FUNCTION_BLOCK CheckStatusVanHetSysteem
VAR
	//Defenieren van de Xas en functies om deze te manipuleren
	XasDrive: AXIS_REF;
	XasDrivePower: MC_Power;
	DePositieVanDeXas AT %I* : LREAL;
	StopDeBoot : MC_Stop;
	VeranderDriveOperationMode : MC_WriteDriveOperationMode;
	OutDeurslot   AT %Q* : BOOL;
	
	//Inputs Vanuit HMI en Variabele voor checken van drive status
	StatusVanDePower : (Uit, Actief, Error );
	KnopDriveAan2 AT %I* : BOOL;
	KnopDriveUit  AT %I* : BOOL;
	IndicatieDriveIsActief   AT %Q* : BOOL;
	KnopStopKnop AT %I* : BOOL;	
	KnopDoorgaan AT %I* : BOOL;	
	
	//Variabele voor het bepalen van de state van het systeem
	StatusVanDeStateVanHetSysteem : (Uit, Joggen, Locatie, Torque);
	KnopJoggModus AT %I* : BOOL;
	KnopLocatieModus  AT %I* : BOOL;
	KnopTorqueControl AT %I* : BOOL;
	IndicatieStatusIsUit   AT %Q* : BOOL;
	IndicatieStatusIsJoggen   AT %Q* : BOOL;
	IndicatieStatusIsLocatie   AT %Q* : BOOL;
	IndicatieStatusIsTorque   AT %Q* : BOOL;
	
	// variabele voor Jogg state
	XasJoggModusFB : MC_MoveVelocity;
	HetTypeJog : (LinksTraag, LinksSnel, RechtsSnel, RechtsTraag, StilStaan);
	KnopJoggModusLinksTraag AT %I* : BOOL;
	KnopJoggModusLinksSnel AT %I* : BOOL;
	KnopJoggModusRechtsTraag AT %I* : BOOL;
	KnopJoggModusRechtsSnel AT %I* : BOOL;
	
	// Variabele voor Locatie state
	XasLocatieModeFB : MC_MoveAbsolute;
	StatusLocatieStatemachine : (WachtenOpNieuweLocatie, Uitvoeren, Bezig, Klaar,Pauzen);
 	DeIngevoerdeTargetPositie AT %I* : LREAL;
	NogAfTeLeggenAfstand AT %Q* : LREAL;
	KnopLocatieUitvoeren AT %I* : BOOL;
	KlaarMetBewegen : BOOL :=FALSE ;
	
	//Variabele voor Torque control
	StatusTorqueStatemachine : (WachtenOpNieuwDoel, Bezig2, Stop);
	DOTorqueDing : MC_TorqueControl;
	DeIngevoerdeTorqueDoel AT %I* : LREAL;
	KnopHervatTorquecontrol AT %I* : BOOL;	
	
	// hoopelijk gelinkde I/O
	InputSensor1 AT %I* : BOOL;
	OutputSysteemIsActiefDeurslot AT %Q* : BOOL;
	SlotDicht: BOOL :=FALSE ;
	SlotOpen: BOOL :=TRUE ;
END_VAR

CheckDrivePower();
CheckStateVanHetSysteem();
	CASE StatusVanDeStateVanHetSysteem OF
		Uit:
			IndicatieStatusIsUit:=TRUE;
			IndicatieStatusIsJoggen:=FALSE;
			IndicatieStatusIsLocatie:=FALSE;
			IndicatieStatusIsTorque:=FALSE;
			OutputSysteemIsActiefDeurslot:=SlotDicht;
		Joggen:
			IndicatieStatusIsUit:=FALSE;
			IndicatieStatusIsJoggen:=TRUE;
			IndicatieStatusIsLocatie:=FALSE;
			IndicatieStatusIsTorque:=FALSE;
			DoJogStatemachine();
			OutputSysteemIsActiefDeurslot:=SlotOpen;
		Locatie:
			NogAfTeLeggenAfstand:= DeIngevoerdeTargetPositie - DePositieVanDeXas;
			IndicatieStatusIsUit:=FALSE;
			IndicatieStatusIsJoggen:=FALSE;
			IndicatieStatusIsLocatie:=TRUE;
			IndicatieStatusIsTorque:=FALSE;
			DoLocatieStatemachine();
			OutputSysteemIsActiefDeurslot:=SlotDicht;		
		Torque:
			NogAfTeLeggenAfstand:= DeIngevoerdeTargetPositie - DePositieVanDeXas;
			IndicatieStatusIsUit:=FALSE;
			IndicatieStatusIsJoggen:=FALSE;
			IndicatieStatusIsLocatie:=FALSE;
			IndicatieStatusIsTorque:=TRUE;
			DoTorqueStatemachine();
			OutputSysteemIsActiefDeurslot:=SlotDicht;
	END_CASE

ACTION CheckDrivePower:
	XasDrivePower
	(
    Axis:= XasDrive,
    Enable:= FALSE,
    Enable_Positive:= TRUE,
    Enable_Negative:= TRUE,
    Override:= 100,
    BufferMode:= ,
    Options:= ,
    Status=> ,
    Busy=> ,
    Active=> ,
    Error=> ,
    ErrorID=> 
	);
//Power Inputs
IF KnopDriveAan2 THEN
	StatusVanDePower:= Actief;
	IndicatieDriveIsActief:=TRUE;
	SetPowerHighElkeKant();
	OutDeurslot:= TRUE;//Deur open
	
END_IF
IF NOT IndicatieDriveIsActief THEN
	StatusVanDePower:=Uit;
	SetPowerLow();
	OutDeurslot:= FALSE;// Deur gesloten
END_IF

//evtueel error checken
END_ACTION

ACTION CheckStateVanHetSysteem:

	VeranderDriveOperationMode
(	Execute:=FALSE,
	DriveOperationMode:=DriveOperationMode_Torque,
	Options:=,
	Axis:=XasDrive,
	Done=>,
	Busy=>,
	Error=>,
	ErrorID=>,);


IF KnopJoggModus AND NOT KnopLocatieModus AND IndicatieDriveIsActief AND NOT KnopTorqueControl THEN
	StatusVanDeStateVanHetSysteem:=Joggen;
	VeranderDriveOperationMode
(	Execute:=TRUE,
	DriveOperationMode:=DriveOperationMode_Default,
	Options:=,
	Axis:=XasDrive,
	Done=>,
	Busy=>,
	Error=>,
	ErrorID=>,);
END_IF

IF NOT KnopJoggModus AND NOT KnopLocatieModus AND IndicatieDriveIsActief AND KnopTorqueControl THEN
	StatusVanDeStateVanHetSysteem:=Torque;
	VeranderDriveOperationMode
(	Execute:=TRUE,
	DriveOperationMode:=DriveOperationMode_Torque,
	Options:=,
	Axis:=XasDrive,
	Done=>,
	Busy=>,
	Error=>,
	ErrorID=>,);

END_IF

IF NOT KnopJoggModus AND  KnopLocatieModus AND IndicatieDriveIsActief AND NOT KnopTorqueControl THEN
	StatusVanDeStateVanHetSysteem:=Locatie;
		
	VeranderDriveOperationMode
(	Execute:=TRUE,
	DriveOperationMode:=DriveOperationMode_Default,
	Options:=,
	Axis:=XasDrive,
	Done=>,
	Busy=>,
	Error=>,
	ErrorID=>,);
END_IF
IF NOT IndicatieDriveIsActief OR  NOT KnopJoggModus AND NOT KnopLocatieModus AND NOT KnopTorqueControl THEN
	StatusVanDeStateVanHetSysteem:=Uit;
	
	VeranderDriveOperationMode
(	Execute:=TRUE,
	DriveOperationMode:=DriveOperationMode_Default,
	Options:=,
	Axis:=XasDrive,
	Done=>,
	Busy=>,
	Error=>,
	ErrorID=>,);
END_IF
END_ACTION

ACTION DoJogStatemachine:
XasJoggModusFB
	(
    Axis:= XasDrive,
	Direction:= 1,
	Velocity :=0 ,
	Execute:=FALSE,
	Deceleration:=0,
	Acceleration :=0,
	Jerk:= ,
	BufferMode:= ,
	Options := ,
	InVelocity => ,
	Active => ,
	Busy => ,
	CommandAborted => ,
	Error => ,
	ErrorID => ,
	);
	
	IF KnopJoggModusLinksTraag THEN
		HetTypeJog:=LinksTraag;
	END_IF
	IF KnopJoggModusLinksSnel THEN
		HetTypeJog:=LinksSnel;
	END_IF
	IF KnopJoggModusRechtsTraag THEN
		HetTypeJog:=RechtsTraag;
	END_IF
	IF KnopJoggModusRechtsSnel THEN
		HetTypeJog:=RechtsSnel;
	END_IF
	IF NOT KnopJoggModusLinksTraag AND NOT KnopJoggModusLinksSnel AND NOT KnopJoggModusRechtsTraag AND NOT KnopJoggModusRechtsSnel THEN
		HetTypeJog:=StilStaan;
	END_IF
	
CASE HetTypeJog OF
	StilStaan:
XasJoggModusFB
(
	Axis:= XasDrive,
	Direction:= 1,
	Velocity :=0 ,
	Execute:=TRUE,
	Deceleration:=0,
	Acceleration :=0,
	Jerk:= ,
	BufferMode:= ,
	Options := ,
	InVelocity => ,
	Active => ,
	Busy => ,
	CommandAborted => ,
	Error => ,
	ErrorID => ,
	);
		LinksTraag:
XasJoggModusFB
(
    Axis:= XasDrive,
	Direction:= MC_Positive_Direction ,
	Velocity :=250 ,
	Execute:=TRUE,
	Deceleration:=0,
	Acceleration :=0,
	Jerk:= ,
	BufferMode:= ,
	Options := ,
	InVelocity => ,
	Active => ,
	Busy => ,
	CommandAborted => ,
	Error => ,
	ErrorID => ,
	);
		LinksSnel:
XasJoggModusFB
(
    Axis:= XasDrive,
	Direction:= MC_Positive_Direction ,
	Velocity :=500 ,
	Execute:=TRUE,
	Deceleration:=0,
	Acceleration :=0,
	Jerk:= ,
	BufferMode:= ,
	Options := ,
	InVelocity => ,
	Active => ,
	Busy => ,
	CommandAborted => ,
	Error => ,
	ErrorID => ,
	);
		RechtsSnel:
XasJoggModusFB
(
    Axis:= XasDrive,
	Direction:= MC_Negative_Direction,
	Velocity :=500 ,
	Execute:=TRUE,
	Deceleration:=0,
	Acceleration :=0,
	Jerk:= ,
	BufferMode:= ,
	Options := ,
	InVelocity => ,
	Active => ,
	Busy => ,
	CommandAborted => ,
	Error => ,
	ErrorID => ,
	);
	
	
	RechtsTraag:
XasJoggModusFB
(
    Axis:= XasDrive,
	Direction:= MC_Negative_Direction,
	Velocity :=250,
	Execute:=TRUE,
	Deceleration:=0,
	Acceleration :=0,
	Jerk:= ,
	BufferMode:= ,
	Options := ,
	InVelocity => ,
	Active => ,
	Busy => ,
	CommandAborted => ,
	Error => ,
	ErrorID => ,
	);

END_CASE
END_ACTION

ACTION DoLocatieStatemachine:

		XasLocatieModeFB
(   Axis:= XasDrive,
	Execute:=FALSE,
	Position := 0,
	Velocity :=0 ,
	Deceleration:=0,
	Acceleration :=0,
	Jerk:= ,
	BufferMode:= ,
	Options := ,
	Done => KlaarMetBewegen,
	Active => ,
	Busy => ,
	CommandAborted => ,
	Error => ,
	ErrorID => , );
		StopDeBoot
(	Axis:= XasDrive,
	Execute:=FALSE,
	Deceleration:=0,
	Jerk:=0,
	Done=>,
	Busy=>,
	Active=>,
	CommandAborted=>,
	Error=>,
	ErrorID=>,);
IF KnopStopKnop THEN
	StatusLocatieStatemachine := Pauzen;
END_IF

CASE StatusLocatieStatemachine OF 
	WachtenOpNieuweLocatie:
	IF KnopLocatieUitvoeren THEN
		StatusLocatieStatemachine:= Uitvoeren;
	END_IF
	Uitvoeren:
	XasLocatieModeFB
(	Axis:= XasDrive,
	Execute:=TRUE,
	Position := DeIngevoerdeTargetPositie,
	Velocity :=500 ,
	Deceleration:=0,
	Acceleration :=0,
	Jerk:= ,
	BufferMode:= ,
	Options := ,
	Done => KlaarMetBewegen,
	Active => ,
	Busy => ,
	CommandAborted => ,
	Error => ,
	ErrorID => , );
	StatusLocatieStatemachine:= Bezig;
	
	Bezig:
	IF KlaarMetBewegen THEN
		StatusLocatieStatemachine:= Klaar;
	END_IF
	Klaar:
		KlaarMetBewegen:=FALSE;
		XasLocatieModeFB
(   Axis:= XasDrive,
	Execute:=FALSE,
	Position := DeIngevoerdeTargetPositie,
	Velocity :=500 ,
	Deceleration:=0,
	Acceleration :=0,
	Jerk:= ,
	BufferMode:= ,
	Options := ,
	Done => KlaarMetBewegen,
	Active => ,
	Busy => ,
	CommandAborted => ,
	Error => ,
	ErrorID => , );
	StatusLocatieStatemachine:= WachtenOpNieuweLocatie;	
		
	Pauzen:
	StopDeBoot
(	Axis:= XasDrive,
	Execute:=TRUE,
	Deceleration:=0,
	Jerk:=0,
	Done=>,
	Busy=>,
	Active=>,
	CommandAborted=>,
	Error=>,
	ErrorID=>,);
	IF KnopDoorgaan THEN
		StatusLocatieStatemachine:= WachtenOpNieuweLocatie;	
	END_IF


END_CASE
END_ACTION

ACTION DoTorqueStatemachine:

		StopDeBoot
(	Axis:= XasDrive,
	Execute:=FALSE,
	Deceleration:=0,
	Jerk:=0,
	Done=>,
	Busy=>,
	Active=>,
	CommandAborted=>,
	Error=>,
	ErrorID=>,);

IF KnopHervatTorquecontrol THEN
	StatusTorqueStatemachine:=Bezig2;
END_IF
	
IF KnopStopKnop THEN
	StatusTorqueStatemachine:=Stop;
END_IF

CASE StatusTorqueStatemachine OF
	WachtenOpNieuwDoel:
		IF KnopHervatTorquecontrol THEN
				StatusTorqueStatemachine:=Bezig2;
		END_IF
	Bezig2:
	
	DOTorqueDing(
	Axis:=XasDrive , 
	Execute:=TRUE , 
	ContinuousUpdate:=TRUE , 
	Relative:=FALSE , 
	Torque:=DeIngevoerdeTorqueDoel, 
	TorqueRamp:=0, 
	VelocityLimitHigh:=1000, 
	VelocityLimitLow:=-1000, 
	BufferMode:= , 
	Options:= , 
	InTorque=> , 
	Busy=> , 
	Active=> , 
	CommandAborted=> , 
	Error=> , 
	ErrorId=> );
	
	Stop:
		StopDeBoot
		(	Axis:= XasDrive,
			Execute:=TRUE,
			Deceleration:=0,
			Jerk:=0,
			Done=>,
			Busy=>,
			Active=>,
			CommandAborted=>,
			Error=>,
			ErrorID=>,);
	END_CASE
END_ACTION

ACTION SetPowerHighElkeKant:
	XasDrivePower
	(
    Axis:= XasDrive,
    Enable:= TRUE,
    Enable_Positive:= TRUE,
    Enable_Negative:= TRUE,
    Override:= 100,
    BufferMode:= ,
    Options:= ,
    Status=> ,
    Busy=> ,
    Active=> ,
    Error=> ,
    ErrorID=> 
	);
END_ACTION

ACTION SetPowerLow:
	XasDrivePower
	(
    Axis:= XasDrive,
    Enable:= FALSE,
    Enable_Positive:= FALSE,
    Enable_Negative:= FALSE,
    Override:= 100,
    BufferMode:= ,
    Options:= ,
    Status=> ,
    Busy=> ,
    Active=> ,
    Error=> ,
    ErrorID=> 
	);
END_ACTION

END_FUNCTION_BLOCK

(* stored: Version 1.1.0.1, ProductVersion 3.1.4024.12
   POU CheckStatusVanHetSysteem: Id {a83cec7a-26ee-4175-ab5a-2ff697203d06}, SpecialFunc None
   Action CheckDrivePower: Id {cbeb062d-b332-4dc4-ab1f-f4bb58083a3a}
   Action CheckStateVanHetSysteem: Id {551ec0e0-108b-48b7-8c88-ecc8de7ea2fb}
   Action DoJogStatemachine: Id {43de3663-3354-4f32-94b3-a1e931bf0c43}
   Action DoLocatieStatemachine: Id {75aa7120-2f71-4f92-bb23-1311f1746a18}
   Action DoTorqueStatemachine: Id {e6f4eca0-fa40-464f-b2a9-0fbcc4d1e4c5}
   Action SetPowerHighElkeKant: Id {640a068c-1238-4885-b710-0a9a6082115d}
   Action SetPowerLow: Id {9f9dfc77-d53a-416c-a4ad-f810d7ff3421} *)
